(* IEC 61131-3 sources: 2026_Projet_YGO_ExcavatriceDragage/TOOLS/TEST_AUTO_CI/RESULTS/DIAG_RESEAUX/tests, 3 files *)

(* ---- test_fb_diag_canopen.st ---- *)
SETUP
VAR
    FB : FB_Diag_CanOpen;
END_VAR
END_SETUP

TEST 'CanOpen : Enable=FALSE desactive le diagnostic'
    FB(Enable := FALSE, CANbusStateRaw := 2, DeviceJoystickStateRaw := DEVICE_STATE.RUNNING);
    ASSERT_FALSE(FB.Ready, 'Ready doit etre FALSE sans Enable');
    ASSERT_EQ(FB.State, E_Diag_State.DISABLED, 'State doit etre DISABLED sans Enable');
END_TEST

TEST 'CanOpen : Enable=TRUE et Bus OK -> Ready et State=READY'
    FB(Enable := TRUE, CANbusStateRaw := 2, DeviceJoystickStateRaw := DEVICE_STATE.RUNNING, SimBypassActive := FALSE, NetworkBypassActive := FALSE);
    ASSERT_TRUE(FB.Ready, 'Ready doit etre TRUE avec Enable');
    ASSERT_EQ(FB.State, E_Diag_State.READY, 'State doit etre READY quand bus et esclave OK');
    ASSERT_FALSE(FB.Error, 'Aucune erreur attendue');
END_TEST

(* ---- test_fb_diag_ethercat.st ---- *)
SETUP
VAR
    FB : FB_Diag_Ethercat;
END_VAR
END_SETUP

TEST 'Ethercat : Enable=FALSE desactive le diagnostic'
    FB(Enable := FALSE, DeviceVariateurStateRaw := DEVICE_STATE.RUNNING, DeviceEncoderM1StateRaw := DEVICE_STATE.RUNNING, DeviceEncoderM2StateRaw := DEVICE_STATE.RUNNING);
    ASSERT_FALSE(FB.Ready, 'Ready doit etre FALSE sans Enable');
    ASSERT_EQ(FB.State, E_Diag_State.DISABLED, 'State doit etre DISABLED sans Enable');
END_TEST

TEST 'Ethercat : Enable=TRUE et Esclaves OK -> Ready et State=READY'
    FB(Enable := TRUE, DeviceVariateurStateRaw := DEVICE_STATE.RUNNING, DeviceEncoderM1StateRaw := DEVICE_STATE.RUNNING, DeviceEncoderM2StateRaw := DEVICE_STATE.RUNNING, DeviceVariateurSimBypass := FALSE, DeviceEncoderM1SimBypass := FALSE, DeviceEncoderM2SimBypass := FALSE, NetworkBypassActive := FALSE);
    ASSERT_TRUE(FB.Ready, 'Ready doit etre TRUE avec Enable');
    ASSERT_EQ(FB.State, E_Diag_State.READY, 'State doit etre READY quand tout est OK');
    ASSERT_FALSE(FB.Error, 'Aucune erreur attendue');
END_TEST

(* ---- test_fb_diag_ihmheartbeat.st ---- *)
SETUP
VAR
    FB : FB_Diag_IhmHeartbeat;
END_VAR
END_SETUP

TEST 'IhmHeartbeat : Enable=FALSE desactive la surveillance'
    FB(Enable := FALSE, TglHeartbeatIhm := FALSE);
    ASSERT_FALSE(FB.HeartbeatIhmOk, 'HeartbeatIhmOk doit etre FALSE');
    ASSERT_TRUE(FB.HeartbeatIhmTimeout, 'HeartbeatIhmTimeout doit etre TRUE');
END_TEST

TEST 'IhmHeartbeat : Front recu -> HeartbeatIhmOk=TRUE'
    FB(Enable := TRUE, TglHeartbeatIhm := FALSE);
    FB(Enable := TRUE, TglHeartbeatIhm := TRUE);
    ASSERT_TRUE(FB.HeartbeatIhmOk, 'HeartbeatIhmOk doit etre TRUE suite au front');
    ASSERT_FALSE(FB.HeartbeatIhmTimeout, 'Pas de timeout');
END_TEST
